FUNCTION_BLOCK FB_TcMatSimObject
VAR_INPUT
	/// set this flag to write FB input values to the TcComObject's input DataAreas. This will overwrite the mapped input values before module execution. Set to FALSE to read the mapped input values from the TcComObject to the FB.
	bWriteFbInputValues: BOOL := TRUE;
END_VAR
VAR
	/// process image src and dst pointers and sizes
	pDataAreas: POINTER TO ST_TcMatSimObjectDataAreaInfo;
	nDataAreas: UDINT;
	/// global interface pointers
	ipObjSrv: ITComObjectServer;
	/// object interface pointers
	ipTcComObj: ITComObject;
	ipTcCyclic: ITcCyclic;
	ipTcPostCyclic: ITcPostCyclic;
	ipTcAdi: ITcADI;
	/// task interface pointers
	ipTask: ITcTask;
	/// initial parameters
	pInitData: POINTER TO TComInitDataHdr;
	/// hResult of interface calls (0 if no error)
	hResult: HRESULT;
	/// module class ID
	moduleClsId: CLSID;
	/// expected/desired module class ID
	assignedClsId: CLSID;
	bClassIdVerified: BOOL;
	/// flag indicating whether the module instance was created dynamically
	bDynInstance: BOOL;
	/// the object state at the time FB_init was called, FB_exit will try to switch to this state (only if this means to shift down)
	eInitialObjState: TCOM_STATE := TCOM_STATE.TCOM_STATE_INIT;
END_VAR

METHOD PUBLIC AssignClassId
VAR_INPUT
	clsId : CLSID;
END_VAR
assignedClsId := clsId;
bClassIdVerified := false;
END_METHOD

PROPERTY ClassId : CLSID
GET
hResult := ReadModuleClassId();
ClassId := moduleClsId;
END_GET
END_PROPERTY

PROPERTY Error : BOOL
GET
Error := FAILED(hResult);
END_GET
END_PROPERTY

PROPERTY ErrorCode : HRESULT
GET
ErrorCode := hResult;
END_GET
END_PROPERTY

{attribute 'object_name' := 'Execute'}
METHOD Execute : HRESULT
VAR
	nDaIdx: UDINT;
	pCurDataArea: POINTER TO ST_TcMatSimObjectDataAreaInfo;
END_VAR

IF (SUCCEEDED(hResult)) THEN
  hResult := VerifyClassId();
END_IF

IF (SUCCEEDED(hResult) AND State<>TCOM_STATE_OP) THEN
  hResult := Tc2_System.E_HRESULTAdsErr.NOTREADY;
END_IF

// get image pointers
IF (SUCCEEDED(hResult)) THEN
  GetImagePtrs(hResult);
END_IF

// copy inputs
IF (pDataAreas<>0 AND bWriteFbInputValues) THEN
  FOR nDaIdx:=0 TO nDataAreas-1 DO
    IF (FAILED(hResult))THEN
      CONTINUE;
    END_IF
    pCurDataArea := pDataAreas + nDaIdx*SIZEOF(ST_TcMatSimObjectDataAreaInfo);
    IF ((pCurDataArea^.eDataAreaType <> E_TcMatSimDataAreaType.InputDst))THEN
      CONTINUE;
    END_IF
    IF (pCurDataArea^.pModuleProcImg<>0 AND pCurDataArea^.pPlcVar<>0) THEN
      MEMCPY(pCurDataArea^.pModuleProcImg,pCurDataArea^.pPlcVar,pCurDataArea^.nSize);
    ELSE
      hResult := Tc2_System.E_HRESULTAdsErr.NOINTERFACE;
    END_IF
  END_FOR
END_IF

// call cycle update
IF (SUCCEEDED(hResult)) THEN
  IF (ipTcCyclic<>0) THEN
    hResult := ipTcCyclic.CycleUpdate(ipTask:= ipTask, ipCaller:= 0, context:= 0);
  ELSE
    hResult := Tc2_System.E_HRESULTAdsErr.NOINTERFACE;
  END_IF
END_IF

// copy outputs
IF (pDataAreas<>0) THEN
  FOR nDaIdx:=0 TO nDataAreas-1 DO
    IF (FAILED(hResult))THEN
      CONTINUE;
    END_IF
    pCurDataArea := pDataAreas + nDaIdx*SIZEOF(ST_TcMatSimObjectDataAreaInfo);
    IF ((pCurDataArea^.eDataAreaType = E_TcMatSimDataAreaType.OutputSrc) OR NOT bWriteFbInputValues) THEN
      IF (pCurDataArea^.pModuleProcImg<>0 AND pCurDataArea^.pPlcVar<>0) THEN
        MEMCPY(pCurDataArea^.pPlcVar,pCurDataArea^.pModuleProcImg,pCurDataArea^.nSize);
      ELSE
        hResult := Tc2_System.E_HRESULTAdsErr.NOINTERFACE;
      END_IF
    END_IF
  END_FOR
END_IF


// call post cyclic update
IF (SUCCEEDED(hResult)) THEN
  IF (ipTcPostCyclic<>0) THEN
    hResult := ipTcPostCyclic.PostCyclicUpdate(ipTask:= 0, ipCaller:= 0, context:= 0);
  ELSE
    hResult := Tc2_System.E_HRESULTAdsErr.NOINTERFACE;
  END_IF
END_IF

ReleaseImagePtrs();

Execute := hResult;
END_METHOD

{attribute 'object_name' := 'FB_exit'}
METHOD FB_exit : BOOL
VAR_INPUT
	/// Online Change
	bInCopyCode: BOOL;
END_VAR

IF (NOT bInCopyCode) THEN
  IF (ipObjSrv<>0) THEN
    ipObjSrv.TcRelease();
    ipObjSrv := 0;
  END_IF

  ReleaseTcComInterface();
END_IF
END_METHOD

{attribute 'object_name' := 'FB_init'}
METHOD FB_init : BOOL
VAR_INPUT
	/// init retain variables
	bInitRetains: BOOL;
	/// Online Change
	bInCopyCode: BOOL;
	oid: OTCID;
END_VAR

FB_init := SUCCEEDED(Init(oid));
END_METHOD

{attribute 'object_name' := 'GetImagePtrs'}
METHOD PRIVATE GetImagePtrs
VAR_INPUT
	hr: REFERENCE TO HRESULT;
END_VAR
VAR
	nDaIdx: UDINT;
	pCurDataArea: POINTER TO ST_TcMatSimObjectDataAreaInfo;
END_VAR

IF (ipTcAdi=0) THEN
  hr := Tc2_System.E_HRESULTAdsErr.NOINTERFACE;
END_IF
IF(State<>TCOM_STATE_OP)THEN
  hr := Tc2_System.E_HRESULTAdsErr.INVALIDSTATE;
END_IF


// get pointers to process images
IF (pDataAreas<>0) THEN
  FOR nDaIdx:=0 TO nDataAreas-1 DO
    pCurDataArea := pDataAreas + nDaIdx*SIZEOF(ST_TcMatSimObjectDataAreaInfo);
    IF (FAILED(hr))THEN
      CONTINUE;
    END_IF
    IF ((pCurDataArea^.eDataAreaType <> E_TcMatSimDataAreaType.InputDst) AND (pCurDataArea^.eDataAreaType <> E_TcMatSimDataAreaType.OutputSrc))THEN
      CONTINUE;
    END_IF
    IF (pCurDataArea^.pModuleProcImg=0 AND pCurDataArea^.nSize>0) THEN
      hr := ipTcAdi.GetImagePtr(size:= pCurDataArea^.nSize , offs:=0 , adi_x:=pCurDataArea^.nDataAreaId , ppData:=ADR(pCurDataArea^.pModuleProcImg));
    END_IF
  END_FOR
END_IF

IF (FAILED(hr)) THEN
  ReleaseImagePtrs();
END_IF
END_METHOD

{attribute 'object_name' := 'GetObjPara'}
METHOD GetObjPara : HRESULT
VAR_INPUT
	pid: PTCID;
	nData: UDINT;
	pData: PVOID;
END_VAR

IF (ipTcComObj=0) THEN
  GetObjPara := Tc2_System.E_HRESULTAdsErr.NOINTERFACE;
END_IF

IF (SUCCEEDED(GetObjPara)) THEN
  GetObjPara := ipTcComObj.TcGetObjPara(pid:=pid,nData,pData,0);
END_IF
END_METHOD

{attribute 'object_name' := 'Init'}
METHOD PROTECTED Init : HRESULT
VAR_INPUT
	oid: OTCID;
END_VAR

// preinitialize variables
memset(ADR(moduleClsId),0,SIZEOF(moduleClsId));
bClassIdVerified := FALSE;
hResult := Tc2_System.E_HRESULTAdsErr.HRESULT_ADS_NOERROR;

// get object server
IF (ipObjSrv=0) THEN
  hResult := FW_ObjMgr_GetObjectServer(_AppInfo.ObjId,ADR(ipObjSrv));
END_IF

// try to get object interfaces
IF (SUCCEEDED(hresult)) THEN
  QueryTcComInterface(hResult,oid);
END_IF

// verify class id
IF (SUCCEEDED(hresult)) THEN
  hresult := VerifyClassId();
END_IF

// query interfaces, if the current state is higher than INIT
IF (SUCCEEDED(hresult) AND State>TCOM_STATE.TCOM_STATE_INIT) THEN
  QueryObjInterfaces(hResult);
END_IF

// return value
Init := hresult;
END_METHOD

{attribute 'object_name' := 'InitObjName'}
METHOD PRIVATE InitObjName
VAR_INPUT
	hr: REFERENCE TO HRESULT;
END_VAR
VAR
	objectName: STRING(255) := 'TempContr_PlcRtFbInstance';
	oid: OTCID;
END_VAR

IF (SUCCEEDED(hr)) THEN
  hr := ipTcComObj.TcGetObjectId(oid);
END_IF

IF (SUCCEEDED(hr) and bDynInstance) THEN
  objectName := TC2_STANDARD.CONCAT(objectName,'_');
  objectName := TC2_STANDARD.CONCAT(objectName,UDINT_TO_STRING(oid));
  hr := ipTcComObj.TcSetObjectName(ADR(objectName));
END_IF
END_METHOD

{attribute 'object_name' := 'Internal_SetObjState'}
METHOD PROTECTED Internal_SetObjState
VAR_INPUT
	hr: REFERENCE TO HRESULT;
	nextState: TCOM_STATE;
END_VAR

// verify class id
IF (SUCCEEDED(hr)) THEN
  hr := VerifyClassId();
END_IF

// switch object state
IF (SUCCEEDED(hr) AND nextState>=TCOM_STATE_INIT) THEN
  IF (ipTcComObj=0) THEN
    hr := Tc2_System.E_HRESULTAdsErr.NOINTERFACE;
  END_IF
  IF (ipObjSrv=0) THEN
    hr := Tc2_System.E_HRESULTAdsErr.NOINTERFACE;
  END_IF
  IF (SUCCEEDED(hr)) THEN
    hr := ipTcComObj.TcSetObjState(nextState,ipObjSrv,pInitData);
  END_IF
END_IF
END_METHOD

{attribute 'object_name' := 'QueryObjInterface'}
METHOD PRIVATE QueryObjInterface
VAR_INPUT
	hr: REFERENCE TO HRESULT;
	iid: REFERENCE TO IID;
	pipItf: POINTER TO ITcUnknown;
END_VAR
VAR CONSTANT
	pNull: PVOID := 0;
END_VAR

IF (SUCCEEDED(hr)) THEN
  IF (ipTcComObj=0) THEN
    hr := Tc2_System.E_HRESULTAdsErr.NOINTERFACE;
  ELSIF (pipItf^=ULINT_TO_DWORD(pNull)) THEN
    hr := ipTcComObj.TcQueryInterface(iid:= iid, pipItf:=pipItf);
  END_IF
END_IF
END_METHOD

{attribute 'object_name' := 'QueryObjInterfaces'}
METHOD PRIVATE QueryObjInterfaces
VAR_INPUT
	hr: REFERENCE TO HRESULT;
END_VAR

IF(State<TCOM_STATE_PREOP)THEN
  hr := Tc2_System.E_HRESULTAdsErr.INVALIDSTATE;
END_IF

//cyclic interface
QueryObjInterface(hr,IID_ITCCYCLIC,ADR(ipTcCyclic));
//post cyclic interface
QueryObjInterface(hr,IID_ITCPOSTCYCLIC,ADR(ipTcPostCyclic));
//adi interface
QueryObjInterface(hr,IID_ITcADI,ADR(ipTcAdi));
END_METHOD

{attribute 'object_name' := 'QueryTcComInterface'}
METHOD PRIVATE QueryTcComInterface
VAR_INPUT
	hr: REFERENCE TO HRESULT;
	oid: OTCID;
END_VAR

IF (ipObjSrv=0) THEN
  hr := Tc2_System.E_HRESULTAdsErr.NOINTERFACE;
END_IF

IF (SUCCEEDED(hr) AND ipTcComObj=0) THEN
  bDynInstance := FALSE;
  IF(oid>0) THEN
    // query interface of existing object
    hr := ipObjSrv.TcQueryObjectInterface(oid,IID_ITComObject,ADR(ipTcComObj));
  ELSE
    // create new instance and get the object interface
    hr := ipObjSrv.TcCreateInstance(assignedClsId,IID_ITComObject,ADR(ipTcComObj));
    IF (SUCCEEDED(hr)) THEN
      bDynInstance := TRUE;
      hr := ipTcComObj.TcSetObjectId(OTCID_CreateNewId);
    END_IF
  END_IF
  IF (SUCCEEDED(hr)) THEN
    eInitialObjState := State;
  END_IF
END_IF
END_METHOD

{attribute 'object_name' := 'ReadModuleClassId'}
METHOD PRIVATE ReadModuleClassId : HRESULT
VAR
	emptyClsId: CLSID;
END_VAR
memset(ADR(emptyClsId),0,SIZEOF(emptyClsId));
IF (memcmp(ADR(moduleClsId),ADR(emptyClsId),SIZEOF(moduleClsId))=0) THEN
  IF (ipTcComObj=0) THEN
    ReadModuleClassId := Tc2_System.E_HRESULTAdsErr.NOINTERFACE;
  END_IF

  //objectClsId := clsid;
  IF (SUCCEEDED(ReadModuleClassId)) THEN
    ReadModuleClassId := ipTcComObj.GetClassId(moduleClsId);
  END_IF
END_IF
END_METHOD

{attribute 'object_name' := 'ReleaseImagePtrs'}
METHOD PRIVATE ReleaseImagePtrs : HRESULT
VAR
	nDaIdx: UDINT;
	pCurDataArea: POINTER TO ST_TcMatSimObjectDataAreaInfo;
END_VAR

IF (ipTcAdi=0) THEN
  ReleaseImagePtrs := Tc2_System.E_HRESULTAdsErr.NOINTERFACE;
END_IF

IF (SUCCEEDED(ReleaseImagePtrs) AND pDataAreas<>0) THEN
  // release pointers to the simulink module process images
  FOR nDaIdx:=0 TO nDataAreas-1 DO
    pCurDataArea := pDataAreas + nDaIdx*SIZEOF(ST_TcMatSimObjectDataAreaInfo);

    IF (pCurDataArea^.pModuleProcImg<>0) THEN
      ipTcAdi.ReleaseImagePtr(pData:=pCurDataArea^.pModuleProcImg);
      pCurDataArea^.pModuleProcImg := 0;
    END_IF
  END_FOR
END_IF
END_METHOD

{attribute 'object_name' := 'ReleaseObjInterfaces'}
METHOD PRIVATE ReleaseObjInterfaces : HRESULT

// release interface pointers
IF (ipTcCyclic<>0) THEN
  ipTcCyclic.TcRelease();
  ipTcCyclic := 0;
END_IF
IF (ipTcPostCyclic<>0) THEN
  ipTcPostCyclic.TcRelease();
  ipTcPostCyclic := 0;
END_IF
IF (ipTcAdi<>0) THEN
  ipTcAdi.TcRelease();
  ipTcAdi := 0;
END_IF
END_METHOD

{attribute 'object_name' := 'ReleaseTcComInterface'}
METHOD PRIVATE ReleaseTcComInterface : HRESULT
VAR
	nStateChangeCnt: DINT := 0;
END_VAR

IF (ipTcComObj<>0) THEN
  WHILE (State>eInitialObjState AND nStateChangeCnt<1000) DO
    State := eInitialObjState;
    nStateChangeCnt := nStateChangeCnt+1;
  END_WHILE
  ReleaseObjInterfaces();
  IF (bDynInstance) THEN
    ReleaseTcComInterface := TC3_MODULE.FW_ObjMgr_DeleteInstance(ADR(ipTcComObj));
  ELSE
    ipTcComObj.TcRelease();
  END_IF
  ipTcComObj := 0;
END_IF
END_METHOD

{attribute 'object_name' := 'ResetHresult'}
METHOD ResetHresult
hResult := S_OK;
END_METHOD

{attribute 'object_name' := 'SaveOnlineParametersForInit'}
METHOD SaveOnlineParametersForInit : HRESULT
VAR
	idx: UINT;
	pInitElemHdr: POINTER TO TComInitDataElmHdr;
	pData: PVOID;
	nData: UDINT;
END_VAR
VAR CONSTANT
	nInitDataAlignment: UDINT := 4;
END_VAR
IF (pInitData<>0) THEN
  pInitElemHdr := pInitData + SIZEOF(pInitData^);
  FOR idx:=1 TO pInitData^.uiElmCnt DO
    pData := pInitElemHdr + ULINT_TO_DWORD(SIZEOF(pInitElemHdr^));
    nData := pInitElemHdr^.cbData;
    SaveOnlineParametersForInit := GetObjPara(pInitElemHdr^.indexOffset,nData,pData);
    IF (FAILED(SaveOnlineParametersForInit)) THEN
      RETURN;
    END_IF
    pInitElemHdr := pData + (nInitDataAlignment*((nData + nInitDataAlignment - 1)/nInitDataAlignment));
  END_FOR
ELSE
	SaveOnlineParametersForInit := Tc2_System.E_HRESULTAdsErr.NOTINIT;
END_IF
END_METHOD


METHOD PUBLIC SetDataAreaInfo
VAR_INPUT
  pDataAreas: POINTER TO ST_TcMatSimObjectDataAreaInfo;
  nDataAreas: UDINT;
END_VAR

THIS^.nDataAreas := nDataAreas;
THIS^.pDataAreas := pDataAreas;
END_METHOD


METHOD PUBLIC SetInitDataInfo
VAR_INPUT
  pInitData : POINTER TO TComInitDataHdr;
END_VAR
this^.pInitData := pInitData;
END_METHOD

{attribute 'object_name' := 'SetObjPara'}
METHOD SetObjPara : HRESULT
VAR_INPUT
	pid: PTCID;
	nData: UDINT;
	pData: PVOID;
END_VAR

IF (ipTcComObj=0) THEN
  SetObjPara := Tc2_System.E_HRESULTAdsErr.NOINTERFACE;
END_IF

IF (SUCCEEDED(SetObjPara)) THEN
  SetObjPara := ipTcComObj.TcSetObjPara(pid:=pid,nData,pData,0);
END_IF
END_METHOD

{attribute 'object_name' := 'SetObjState'}
METHOD SetObjState : HRESULT
VAR_INPUT
	finalState: TCOM_STATE;
END_VAR
VAR
	bShiftUp: BOOL;
	bShiftDown: BOOL;
	currentState: TCOM_STATE;
END_VAR

currentState := State;

bShiftUp := finalState>currentState;
bShiftDown := finalState<currentState;

// do not switch up on error
IF (FAILED(hresult)) THEN
  bShiftUp := FALSE;
END_IF
// reset existing error on switching down
IF (bShiftDown) THEN
  ResetHresult();
END_IF

// prepared state switch
CASE currentState OF
  TCOM_STATE_INIT:
    IF(bShiftUp) THEN
      QueryTcComInterface(hResult,0);
      Internal_SetObjState(hResult,TCOM_STATE.TCOM_STATE_PREOP);
      InitObjName(hResult);
    END_IF

  TCOM_STATE_PREOP:
    IF(bShiftUp) THEN
      Internal_SetObjState(hResult,TCOM_STATE.TCOM_STATE_SAFEOP);
      QueryObjInterfaces(hResult);
    ELSIF (bShiftDown) THEN
      Internal_SetObjState(hResult,TCOM_STATE.TCOM_STATE_INIT);
    END_IF

  TCOM_STATE_SAFEOP:
    IF(bShiftUp) THEN
      Internal_SetObjState(hResult,TCOM_STATE.TCOM_STATE_OP);
      QueryObjInterfaces(hResult);
    ELSIF (bShiftDown) THEN
      Internal_SetObjState(hResult,TCOM_STATE.TCOM_STATE_PREOP);
      ReleaseObjInterfaces();
    END_IF


  TCOM_STATE_OP:
    IF (bShiftDown) THEN
      Internal_SetObjState(hResult,TCOM_STATE.TCOM_STATE_SAFEOP);
    END_IF
END_CASE

SetObjState := hResult;
END_METHOD

PROPERTY State : TCOM_STATE
GET
VAR
	hr: HRESULT := S_OK;
	eObjState: TCOM_STATE;
END_VAR

IF (ipTcComObj<>0) THEN
  hr := ipTcComObj.TcGetObjState(ADR(eObjState));
IF (FAILED(hr)) THEN
  eObjState := TCOM_STATE.TCOM_STATE_INIT;
END_IF
ELSE
  eObjState := TCOM_STATE.TCOM_STATE_INIT;
END_IF
State := eObjState;
END_GET
SET
SetObjState(State);
END_SET
END_PROPERTY

{attribute 'object_name' := 'VerifyClassId'}
METHOD PRIVATE VerifyClassId : HRESULT
VAR
	emptyClsId: CLSID;
END_VAR
memset(ADR(emptyClsId),0,SIZEOF(emptyClsId));
IF (bClassIdVerified) THEN
  // class ID was already verified
  VerifyClassId := Tc2_System.E_HRESULTAdsErr.HRESULT_ADS_NOERROR;
ELSIF (memcmp(ADR(assignedClsId),ADR(emptyClsId),SIZEOF(assignedClsId))=0) THEN
  // skip class ID verification if no assignedClsId specified
  VerifyClassId := Tc2_System.E_HRESULTAdsErr.HRESULT_ADS_NOERROR;
ELSE
  // verify class ID
  VerifyClassId := ReadModuleClassId();

  IF (SUCCEEDED(VerifyClassId)) THEN
    IF (memcmp(ADR(assignedClsId),ADR(moduleClsId),SIZEOF(assignedClsId))<>0) THEN
     VerifyClassId := Tc2_System.E_HRESULTAdsErr.INVALIDCLSID;
    END_IF
  END_IF
  bClassIdVerified := SUCCEEDED(VerifyClassId);
END_IF
END_METHOD

END_FUNCTION_BLOCK

(* stored: Version 1.1.0.1, ProductVersion 3.1.4020.12
   POU FB_TcMatSimObject: Id {b2572486-ee32-4a5d-a8dc-2597c127d518}, SpecialFunc None
   Method AssignClassId: Id {70aee05c-b7c0-4a1a-90db-a70048b378df}
   Property ClassId: Id {d8ca0918-0e78-4363-b5dd-4f6ed4ff484d}
   Get Get: Id {fb10726a-5fe9-452b-9b6d-0a3a6eb9b2e6}
   Property Error: Id {8e813f4f-7536-4b96-9ed0-d5ec7991eb96}
   Get Get: Id {f19b9680-100e-4e25-a70c-bbedaec48dc7}
   Property ErrorCode: Id {b6dcb6b3-f64f-4d82-a418-e646702ce997}
   Get Get: Id {80dadab1-68fc-485d-a27b-fe4d1567484d}
   Method Execute: Id {4b2e5b40-a87a-4d8e-9d2f-5f4b40c412c3}
   Method FB_exit: Id {9cefef2c-4969-4c6f-a7a6-f930c671b040}
   Method FB_init: Id {b737699c-ef7a-4d97-a9e8-f486dc79ed2d}
   Method GetImagePtrs: Id {e8ac6731-9104-4bbb-82ff-e96a33f0ff3e}
   Method GetObjPara: Id {e5e98eee-5a6c-4a73-965b-dbf7b5ff0c06}
   Method Init: Id {963f3404-4988-4233-8012-c0374a02f102}
   Method InitObjName: Id {fd5d84e2-1534-4e0e-9f4c-969235b7bde0}
   Method Internal_SetObjState: Id {82d4f3a2-6c46-42c7-9dc5-dd617d11dd6e}
   Method QueryObjInterface: Id {c9141cfa-39eb-40aa-b485-bcc9681925b2}
   Method QueryObjInterfaces: Id {15d01b2f-160a-46ea-abff-0f9bfd968949}
   Method QueryTcComInterface: Id {b7d9ad74-23b9-4df2-90a5-e60bca15ceca}
   Method ReadModuleClassId: Id {4430359c-9c39-4c2f-b0ca-4e5015b398ea}
   Method ReleaseImagePtrs: Id {1d264f8c-b8dd-4a11-86da-e80f177d255d}
   Method ReleaseObjInterfaces: Id {7e4811e1-be29-4f78-8346-9346a546acc2}
   Method ReleaseTcComInterface: Id {a43dd200-5b99-4dae-9133-b492e2b0015c}
   Method ResetHresult: Id {264ebbb6-42df-4044-938d-60ac6b8c4f52}
   Method SaveOnlineParametersForInit: Id {436060e4-c64f-4a49-a852-9b372f4a2382}
   Method SetDataAreaInfo: Id {11a4ecef-f4b8-4ea3-b32a-f5c95d2a16a3}
   Method SetInitDataInfo: Id {a4b3eb8c-b58b-4cd6-a9be-95800eb47e3c}
   Method SetObjPara: Id {a2744ffc-3f1e-4a63-933a-1d4138de4f1f}
   Method SetObjState: Id {55da74ca-d54d-41c5-a667-b48e4a25fc1b}
   Property State: Id {66da3436-c568-4814-8054-49fe99c36fa7}
   Get Get: Id {a0f388fb-763d-40a3-8624-0fdda314ac9b}
   Set Set: Id {de12d318-0cfa-45de-978f-154f895a14a5}
   Method VerifyClassId: Id {239bccd7-2f3a-47e3-959e-96b59c3eff01} *)
